FUNCTION_BLOCK FB_TsConnection_EtherCatState_EL1918
VAR_INPUT
    nEtherCATState : UINT; // EtherCAT Slave State
END_VAR
VAR_OUTPUT
    sEtherCATState : STRING;
END_VAR

CASE nEtherCATState OF
    16#0001: sEtherCATState := 'INIT';
    16#0002: sEtherCATState := 'PREOP';
    16#0003: sEtherCATState := 'BOOT';
    16#0004: sEtherCATState := 'SAFEOP';
    16#0008: sEtherCATState := 'OP';
ELSE
    sEtherCATState := 'undefined';
END_CASE

END_FUNCTION_BLOCK

(* stored: Version 1.1.0.1, ProductVersion 3.1.4024.15
   POU FB_TsConnection_EtherCatState_EL1918: Id {d911f51f-b045-4bc2-a239-7afbce64cb11}, SpecialFunc None *)
